INTERFACE ITF_BaseMainComponent_HMI_Connector EXTENDS ITF_BaseComplexElement_HMI_Connector

END_INTERFACE

(* stored: Version 1.1.0.1
   Itf ITF_BaseMainComponent_HMI_Connector: Id {770e6841-0e75-097b-268d-045557e39b52} *)
